TYPE ST_UcWinchControl :
STRUCT
    bDisable          : BOOL; (* Glavni Safety Enable *)
    bManualEnable     : BOOL; (* HMI Manual Mode *)
    bBtn_Dir1         : BOOL; (* Tipka: Slow ili In *)
    bBtn_Dir2         : BOOL; (* Tipka: Fast ili Out *)
    bValve_Dir1       : BOOL; (* Aktivan izlaz 1 *)
    bValve_Dir2       : BOOL; (* Aktivan izlaz 2 *)
    bReq_Pump         : BOOL; (* Pumpa radi *)
    bSts_SystemSafe   : BOOL; (* Zeleno = Safe *)
    bSts_ManualEn     : BOOL; (* Zeleno = Manual *)
END_STRUCT
END_TYPE

(* stored: Version 1.1.0.1, ProductVersion 3.1.4026.17
   DUT ST_UcWinchControl: Id {d4a2d39e-fe96-4b6c-bba1-7a652908d874} *)
